Omron CX-Programmer project 新規ﾌﾟﾛｼﾞｪｸﾄ (CX-Programmer 9.61)

# PLC hoge1: CP1L L

## Program 新規ﾌﾟﾛｸﾞﾗﾑ1 (cyclic task 0)
Local symbols
I 0.00 BOOL
Q 100.00 BOOL

### Section ｾｸｼｮﾝ1

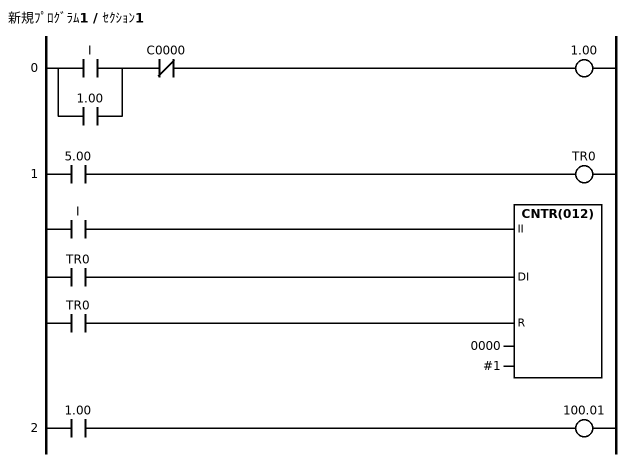
; rung 0
LD I
OR 1.00
ANDNOT C0000
OUT 1.00
; rung 1
LD I
LD 5.00
OUT TR0
LD TR0
CNTR(012) 0000 #1
; rung 2
LD 1.00
OUT 100.01

### Section END
; rung 0
END(001)